Universal Robots PolyScope program: venosa mq estados 4 cam.urp

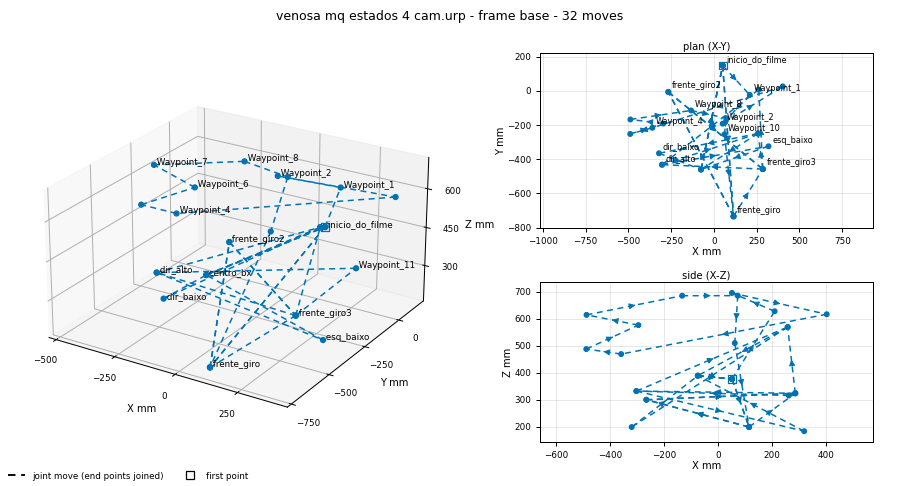
[picture p0: tool path of venosa mq estados 4 cam.urp in frame base, 32 of 32 moves have a stored position in this frame; points joined in program order, loops and branches not executed]
Program venosa mq estados 4 cam (installation=default directory=/programs/usbdisk createdIn=3.10.1.76190 lastSavedIn=3.10.1.76190 robotSerialNumber=2016331323)
Calibrated DH parameters: a=[0.000045, -0.243749, -0.203764, -0.000005, 0.000123, 0]; d=[0.152024, -1.672567, 11.732654, -9.94768, 0.085297, 0.082386]; alpha=[1.569842, 0.003628, 0.006344, 1.57195, -1.572092, 0]; deltaTheta=[0.000055, -0.024957, 0.328359, -0.303533, 0.000075, 0.000016]
BeforeStart
  comm := False
  interrupt := False
  vid_com := [0,0,0]
  Sel := 999
  Start := 999
  video := False
  Loop While (checkContinuously=false) expression=comm≟ False
    comm := socket_open("192.168.99.100",9001)
  Script: socket_send_string("conexao aberta")
Robot Program (runOnlyOnce=false)
  MoveJ speed 60 deg/s, acceleration 80 deg/s^2 (useActiveTCP=true)
    Waypoint inicio_do_filme: TCP in base x=51.208 y=147.993 z=376.683 mm, rx=1.1897 ry=-1.1188 rz=1.2366 rad; joints [98.792, -166.173, 19.211, -37.345, -96.882, -138.028] deg; flange x=47.674 y=351.531 z=418.631 mm, rx=1.4313 ry=-0.5423 rz=0.6241 rad
    Script: socket_send_string("home_0")
    Wait Condition expression=Start≟1 or Start≟2
    If Start≟2
      Folder Danca
        Script: socket_send_string("danca_1")
        Loop While (checkContinuously=true) expression=Start≠0
          MoveJ speed 100 deg/s, acceleration 220 deg/s^2 (useActiveTCP=true)
            Waypoint Waypoint_1: TCP in base x=209.295 y=-23.76 z=627.936 mm, rx=0.0536 ry=-0.3833 rz=0.5202 rad; joints [25.586, -182.4, 88.65, -154.413, -90.664, 229.976] deg; flange x=323.162 y=32.336 z=463.353 mm, rx=0.1944 ry=-0.3308 rz=-0.2551 rad
            Waypoint Waypoint_2: TCP in base x=50.984 y=-192.029 z=695.996 mm, rx=0.4611 ry=-0.1009 rz=0.0738 rad; joints [24.921, -140.097, 106.259, -219.954, -68.232, 201.472] deg; flange x=123.19 y=-99.79 z=524.303 mm, rx=0.4743 ry=0.0849 rz=-0.6963 rad
            Waypoint Waypoint_3: TCP in base x=402.472 y=25.799 z=616.927 mm, rx=-0.0697 ry=-0.0925 rz=0.3622 rad; joints [17.187, -135.525, -41.809, -87.947, -93.999, 228.948] deg; flange x=475.681 y=35.703 z=422.653 mm, rx=-0.0291 ry=-0.1124 rz=-0.4219 rad
            Waypoint Waypoint_4: TCP in base x=-360.047 y=-215.964 z=469.186 mm, rx=0.079 ry=-1.1865 rz=0.2861 rad; joints [17.753, 2.71, -116.283, -88.686, -94.003, 228.949] deg; flange x=-160.208 y=-163.762 z=445.963 mm, rx=0.5289 ry=-1.0702 rz=-0.4044 rad
            Waypoint Waypoint_5: TCP in base x=-489.412 y=-252.244 z=487.887 mm, rx=0.073 ry=-1.1553 rz=0.2787 rad; joints [17.137, 2.694, -78.551, -128.171, -93.991, 228.95] deg; flange x=-289.897 y=-202.079 z=458.266 mm, rx=0.5117 ry=-1.0443 rz=-0.4168 rad
            Waypoint Waypoint_6: TCP in base x=-296.12 y=-191.355 z=576.602 mm, rx=0.0579 ry=-1.0832 rz=0.2879 rad; joints [17.15, -21.94, -102.997, -83.298, -93.994, 228.949] deg; flange x=-99.068 y=-142.519 z=532.045 mm, rx=0.4698 ry=-0.983 rz=-0.4188 rad
            Waypoint Waypoint_7: TCP in base x=-488.569 y=-167.36 z=614.619 mm, rx=-0.0136 ry=-1.2623 rz=0.131 rad; joints [8.254, -35.552, -41.209, -121.068, -93.991, 228.947] deg; flange x=-281.667 y=-148.953 z=607.37 mm, rx=0.4769 ry=-1.188 rz=-0.546 rad
            Waypoint Waypoint_8: TCP in base x=-133.685 y=-114.831 z=685.693 mm, rx=-0.0287 ry=-1.1088 rz=0.1472 rad; joints [8.292, -74.647, -62.125, -69.9, -93.994, 228.943] deg; flange x=69.715 y=-97.233 z=646.726 mm, rx=0.4031 ry=-1.0497 rz=-0.555 rad
            Waypoint Waypoint_9: TCP in base x=72.457 y=-160.105 z=685.924 mm, rx=0.6935 ry=-0.9793 rz=1.2875 rad; joints [81.88, -74.701, -62.13, -69.92, -93.995, 228.945] deg; flange x=113.042 y=39.927 z=646.676 mm, rx=0.9523 ry=-0.5998 rz=0.5937 rad
            Waypoint Waypoint_10: TCP in base x=61.419 y=-254.47 z=510.056 mm, rx=0.7318 ry=-1.0148 rz=1.2772 rad; joints [81.943, -35.981, -123.832, -44.204, -93.737, 228.945] deg; flange x=100.508 y=-52.476 z=480.549 mm, rx=0.9985 ry=-0.617 rz=0.5916 rad
        Script: stopj(2)
        Script: socket_send_string("interromper_danca")
    ElseIf Start≟1
      If Start≠0 (checkContinuously=true)
        interrupt := True
        Switch expression=Sel
          Case (caseValue=1)
            Folder Rotina Video 1
              MoveJ speed 180 deg/s, acceleration 250 deg/s^2 (useActiveTCP=true)
                Script: socket_send_string("start_video_1")
                Waypoint frente_giro: motionParameters(blendRadius=0); TCP in base x=114.529 y=-733.944 z=198.695 mm, rx=1.1286 ry=-1.1446 rz=1.2534 rad; joints [90.394, 3.262, -4.677, -184.263, -90.979, -134.255] deg; flange x=115.651 y=-529.371 z=235.416 mm, rx=1.3863 ry=-0.586 rz=0.6351 rad
                Waypoint frente_giro2: motionParameters(blendRadius=0.05); TCP in base x=-266.69 y=-6.601 z=299.677 mm, rx=1.4295 ry=-0.9647 rz=1.5441 rad; joints [-48.641, -1.485, -24.691, -149.41, 71.438, -136.121] deg; flange x=-345.69 y=180.863 z=342.294 mm, rx=1.5467 ry=-0.3154 rz=0.9503 rad
                Waypoint frente_giro3: TCP in base x=285.848 y=-457.668 z=323.805 mm, rx=0.8532 ry=-1.3147 rz=0.917 rad; joints [-11.57, -143.925, -41.216, -11.685, -12.887, -118.773] deg; flange x=369.13 y=-271.826 z=365.361 mm, rx=1.2385 ry=-0.8521 rz=0.2925 rad
                Waypoint dir_alto: TCP in base x=-303.629 y=-431.898 z=331.906 mm, rx=1.147 ry=-1.3647 rz=2.0179 rad; joints [8.553, -32.921, 38.761, -150.615, 17.6, -136] deg; flange x=-412.468 y=-255.336 z=345.319 mm, rx=1.3941 ry=-0.7246 rz=1.4359 rad
                Waypoint esq_alto: TCP in base x=257.75 y=-249.628 z=569.455 mm, rx=0.6273 ry=-1.5594 rz=1.6399 rad; joints [32.466, -100.522, -51.024, -39.237, -41.525, 270] deg; flange x=256.088 y=-42.664 z=588.516 mm, rx=1.0694 ry=-1.092 rz=1.0357 rad
                Waypoint centro_bx: motionParameters(blendRadius=0.05); TCP in base x=-75.564 y=-459.746 z=388.988 mm, rx=1.2104 ry=-1.0938 rz=1.2402 rad; joints [-81.026, -80.247, -114.352, 18.926, 84.004, -138] deg; flange x=-82.464 y=-256.191 z=430.432 mm, rx=1.4399 ry=-0.5131 rz=0.6273 rad
                Waypoint inicio_do_filme: TCP in base x=51.208 y=147.993 z=376.683 mm, rx=1.1897 ry=-1.1188 rz=1.2366 rad; joints [98.792, -166.173, 19.211, -37.345, -96.882, -138.028] deg; flange x=47.674 y=351.531 z=418.631 mm, rx=1.4313 ry=-0.5423 rz=0.6241 rad
                interrupt := False
                Script: socket_send_string("fim_video_1")
                Wait Condition expression=Start≟0
          Case (caseValue=2)
            Folder Rotina Video 2
              MoveJ speed 180 deg/s, acceleration 250 deg/s^2 (useActiveTCP=true)
                Script: socket_send_string("start_video_2")
                Waypoint frente_giro: motionParameters(blendRadius=0); TCP in base x=114.529 y=-733.944 z=198.695 mm, rx=1.1286 ry=-1.1446 rz=1.2534 rad; joints [90.394, 3.262, -4.677, -184.263, -90.979, -134.255] deg; flange x=115.651 y=-529.371 z=235.416 mm, rx=1.3863 ry=-0.586 rz=0.6351 rad
                Waypoint frente_giro3: TCP in base x=285.848 y=-457.668 z=323.805 mm, rx=0.8532 ry=-1.3147 rz=0.917 rad; joints [-11.57, -143.925, -41.216, -11.685, -12.887, -118.773] deg; flange x=369.13 y=-271.826 z=365.361 mm, rx=1.2385 ry=-0.8521 rz=0.2925 rad
                Waypoint esq_alto: TCP in base x=257.75 y=-249.628 z=569.455 mm, rx=0.6273 ry=-1.5594 rz=1.6399 rad; joints [32.466, -100.522, -51.024, -39.237, -41.525, 270] deg; flange x=256.088 y=-42.664 z=588.516 mm, rx=1.0694 ry=-1.092 rz=1.0357 rad
                Waypoint dir_baixo: motionParameters(blendRadius=0.05); TCP in base x=-321.017 y=-365.217 z=198.414 mm, rx=0.9367 ry=-1.1225 rz=1.8338 rad; joints [-2.971, -32.485, 89.155, -180.73, 24.475, 553.487] deg; flange x=-382.977 y=-167.692 z=179.847 mm, rx=1.1636 ry=-0.6101 rz=1.1836 rad
                Waypoint centro_bx: motionParameters(blendRadius=0.05); TCP in base x=-75.564 y=-459.746 z=388.988 mm, rx=1.2104 ry=-1.0938 rz=1.2402 rad; joints [-81.026, -80.247, -114.352, 18.926, 84.004, -138] deg; flange x=-82.464 y=-256.191 z=430.432 mm, rx=1.4399 ry=-0.5131 rz=0.6273 rad
                Waypoint inicio_do_filme: TCP in base x=51.208 y=147.993 z=376.683 mm, rx=1.1897 ry=-1.1188 rz=1.2366 rad; joints [98.792, -166.173, 19.211, -37.345, -96.882, -138.028] deg; flange x=47.674 y=351.531 z=418.631 mm, rx=1.4313 ry=-0.5423 rz=0.6241 rad
                interrupt := False
                Script: socket_send_string("fim_video_2")
                Wait Condition expression=Start≟0
          Case (caseValue=3)
            Folder Rotina Video 3
              MoveJ speed 180 deg/s, acceleration 250 deg/s^2 (useActiveTCP=true)
                Script: socket_send_string("start_video_3")
                Waypoint frente_giro: motionParameters(blendRadius=0.05); TCP in base x=114.529 y=-733.944 z=198.695 mm, rx=1.1286 ry=-1.1446 rz=1.2534 rad; joints [90.394, 3.262, -4.677, -184.263, -90.979, -134.255] deg; flange x=115.651 y=-529.371 z=235.416 mm, rx=1.3863 ry=-0.586 rz=0.6351 rad
                Waypoint frente_giro2: motionParameters(blendRadius=0.05); TCP in base x=-266.69 y=-6.601 z=299.677 mm, rx=1.4295 ry=-0.9647 rz=1.5441 rad; joints [-48.641, -1.485, -24.691, -149.41, 71.438, -136.121] deg; flange x=-345.69 y=180.863 z=342.294 mm, rx=1.5467 ry=-0.3154 rz=0.9503 rad
                Waypoint frente_giro3: TCP in base x=285.848 y=-457.668 z=323.805 mm, rx=0.8532 ry=-1.3147 rz=0.917 rad; joints [-11.57, -143.925, -41.216, -11.685, -12.887, -118.773] deg; flange x=369.13 y=-271.826 z=365.361 mm, rx=1.2385 ry=-0.8521 rz=0.2925 rad
                Waypoint Waypoint_11: TCP in base x=261.927 y=7.232 z=315.553 mm, rx=0.7766 ry=-1.2189 rz=1.1536 rad; joints [53.936, -192.33, 47.819, -48.838, -71.964, 235.793] deg; flange x=319.02 y=206.808 z=326.042 mm, rx=1.1183 ry=-0.7832 rz=0.503 rad
                Waypoint dir_alto: motionParameters(blendRadius=0.05); TCP in base x=-303.629 y=-431.898 z=331.906 mm, rx=1.147 ry=-1.3647 rz=2.0179 rad; joints [8.553, -32.921, 38.761, -150.615, 17.6, -136] deg; flange x=-412.468 y=-255.336 z=345.319 mm, rx=1.3941 ry=-0.7246 rz=1.4359 rad
                Waypoint esq_baixo: TCP in base x=318.947 y=-324.368 z=183.072 mm, rx=1.0731 ry=-0.8713 rz=0.6999 rad; joints [7.997, -155.808, -71.925, 18.898, -26.152, -136] deg; flange x=397.902 y=-132.164 z=187.981 mm, rx=1.2918 ry=-0.3848 rz=0.0402 rad
                Waypoint centro_bx: motionParameters(blendRadius=0.05); TCP in base x=-75.564 y=-459.746 z=388.988 mm, rx=1.2104 ry=-1.0938 rz=1.2402 rad; joints [-81.026, -80.247, -114.352, 18.926, 84.004, -138] deg; flange x=-82.464 y=-256.191 z=430.432 mm, rx=1.4399 ry=-0.5131 rz=0.6273 rad
                Waypoint inicio_do_filme: TCP in base x=51.208 y=147.993 z=376.683 mm, rx=1.1897 ry=-1.1188 rz=1.2366 rad; joints [98.792, -166.173, 19.211, -37.345, -96.882, -138.028] deg; flange x=47.674 y=351.531 z=418.631 mm, rx=1.4313 ry=-0.5423 rz=0.6241 rad
                interrupt := False
                Script: socket_send_string("fim_video_3")
                Wait Condition expression=Start≟0
      Script: stopj(2)
      If interrupt
        Script: socket_send_string("interromper_video")
Thread Thread_1 (runOnlyOnce=false trackProgramExecution=false)
  vid_com := socket_read_ascii_float(2)
  If vid_com[0]≟2
    Start := vid_com[1]
    Sel := vid_com[2]
    vid_com := [0,0,0]
  Script: sync()
